// SIMATIC S7-200 SMART project (STEP 7-Micro/WIN SMART), CPU ST40

SYMBOL_TABLE 系统符号
Clock_1s         SM0.5    // 针对 1 s 的周期时间，时钟脉冲接通 0.5 s，断开 0.5 s.
END_SYMBOL_TABLE

ORGANIZATION_BLOCK MAIN:OB1
TITLE=程序注释
BEGIN
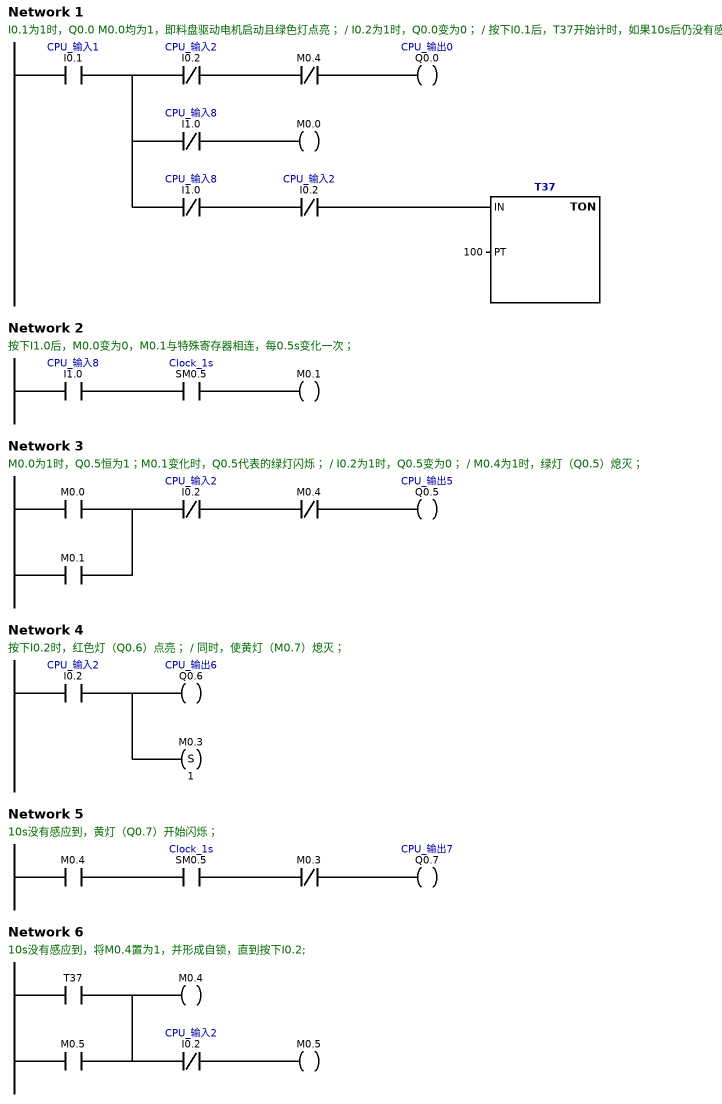
Network 1
// I0.1为1时，Q0.0 M0.0均为1，即料盘驱动电机启动且绿色灯点亮；
// I0.2为1时，Q0.0变为0；
// 按下I0.1后，T37开始计时，如果10s后仍没有感应到货物，则M0.4变为1，此时，发动机（Q0.0）停止工作；
LD     CPU_输入1:I0.1
LPS
AN     CPU_输入2:I0.2
AN     M0.4
=      CPU_输出0:Q0.0
LRD
AN     CPU_输入8:I1.0
=      M0.0
LPP
AN     CPU_输入8:I1.0
AN     CPU_输入2:I0.2
TON    T37, 100
Network 2
// 按下I1.0后，M0.0变为0，M0.1与特殊寄存器相连，每0.5s变化一次；
LD     CPU_输入8:I1.0
A      Clock_1s:SM0.5
=      M0.1
Network 3
// M0.0为1时，Q0.5恒为1；M0.1变化时，Q0.5代表的绿灯闪烁；
// I0.2为1时，Q0.5变为0；
// M0.4为1时，绿灯（Q0.5）熄灭；
LD     M0.0
O      M0.1
AN     CPU_输入2:I0.2
AN     M0.4
=      CPU_输出5:Q0.5
Network 4
// 按下I0.2时，红色灯（Q0.6）点亮；
// 同时，使黄灯（M0.7）熄灭；
LD     CPU_输入2:I0.2
=      CPU_输出6:Q0.6
S      M0.3, 1
Network 5
// 10s没有感应到，黄灯（Q0.7）开始闪烁；
LD     M0.4
A      Clock_1s:SM0.5
AN     M0.3
=      CPU_输出7:Q0.7
Network 6
// 10s没有感应到，将M0.4置为1，并形成自锁，直到按下I0.2;
LD     T37
O      M0.5
=      M0.4
AN     CPU_输入2:I0.2
=      M0.5
END_ORGANIZATION_BLOCK
